// TIA Portal V17 export
// export: Created 2024-09-02T12:50:25.1727323Z, ExportSetting WithDefaults, DisplayName Totally Integrated Automation Portal, DisplayVersion V17, DisplayName TIA Portal Openness, DisplayVersion V17, DisplayName TIA Portal Version Control Interface, DisplayVersion V17, DisplayName STEP 7 Professional, DisplayVersion V17, DisplayName STEP 7 Safety, DisplayVersion V17, DisplayName WinCC Professional, DisplayVersion V17
VAR_GLOBAL   // PLC tag table "Standard-Variablentabelle"
   System_Byte AT %MB1 : Byte;
   FirstScan AT %M1.0 : Bool;
   DiagStatusUpdate AT %M1.1 : Bool;
   AlwaysTRUE AT %M1.2 : Bool;
   AlwaysFALSE AT %M1.3 : Bool;
   Clock_Byte AT %MB0 : Byte;
   Clock_10Hz AT %M0.0 : Bool;
   Clock_5Hz AT %M0.1 : Bool;
   "Clock_2.5Hz" AT %M0.2 : Bool;
   Clock_2Hz AT %M0.3 : Bool;
   "Clock_1.25Hz" AT %M0.4 : Bool;
   Clock_1Hz AT %M0.5 : Bool;
   "Clock_0.625Hz" AT %M0.6 : Bool;
   "Clock_0.5Hz" AT %M0.7 : Bool;
   I_controle_position_of_Pallet AT %I50.6 : Bool;
   Tag_14 AT %ID4000 : DWord;
   I_active_energy AT %I4.0 : LReal;
   I_active_Air AT %ID126 : DWord;
   Q_Energy_Counter_HW_Reset AT %Q6.2 : Bool;
   I_screw_present_OP70_3 AT %I56.4 : Bool;
   test AT %I56.5 : Bool;
   test2 AT %I56.6 : Bool;
   test_3 AT %I56.3 : Bool;
END_VAR
VAR_GLOBAL CONSTANT   // user constants
   SCREEN_SETUP : Word := W#16#0201;
   SCREEN_POWER_UP : Word := W#16#0202;
   SCREEN_UNIT : Word := W#16#0203;
   SCREEN_NUT_RUNNER : Word := W#16#0204;
   SCREEN_NUT_RUNNER_GROUP : Word := W#16#0205;
   SCREEN_CYCLE_TYPES : Word := W#16#0206;
   SCREEN_USER_DEFINE : Word := W#16#0207;
   konst_mds_PRGadr : DInt := 1280;   // Programmfach startadresse
   konst_mds_TAF_adr : DInt := 12640;   // Status TAF start address / Status TAF startadresse
   konst_mds_TAF_max : DInt := 512;   // Status TAF Number maximum / Status TAF Nummer maximal
   konst_mds_PRG_lng : DInt := 222;   // Programmfach länge
   konst_mds_DMC_SollAdr : DInt := 17248;   // DMC SOLL startadresse
   konst_mds_DMC_SollMax : DInt := 18970;   // DMC SOLL max. adresse
   konst_mds_MKmit : DInt := 13152;   // MK mit NA startadresse
   konst_mds_MKohne : DInt := 15200;   // MK ohne NA startadresse
   konst_mds_DMC_IstAdr : DInt := 19012;   // DMC IST startadresse
   konst_mds_SMC_IstMax : DInt := 20962;   // DMC IST max. adresse
   konst_mds_QDAT_adr : DInt := 21012;   // Q-Daten startadresse
   konst_mds_QDAT_max : DInt := 31722;   // Q-Daten max. adresse
   MUSTER_AnwDB_Drucker_GST : Bool := 0;   // ONLY FOR SAMPLE _ REMOVE BY SW CREATION / NUR ZUR MUSTERDARSTELLUNG _ ENTEFERNEN BEI SW ERSTELLUNG
   konst_mds_ANBAUTEILE_Lange : Int := 42;
   konst_mds_DMC_lange : Int := 50;
   UFM_MAX_CONCURRENT_TASKS_LESS_ONE : Int := 9;
   UFM_MAX_LOGLINES : UInt := 99;
END_VAR
